// TIA Portal V17 export
// export: Created 2024-09-02T12:50:26.2822455Z, ExportSetting WithDefaults, DisplayName Totally Integrated Automation Portal, DisplayVersion V17, DisplayName TIA Portal Openness, DisplayVersion V17, DisplayName TIA Portal Version Control Interface, DisplayVersion V17, DisplayName STEP 7 Professional, DisplayVersion V17, DisplayName STEP 7 Safety, DisplayVersion V17, DisplayName WinCC Professional, DisplayVersion V17
TYPE "TypeOperatingModes"
// stored: IsFailsafeCompliant false
   STRUCT
      lamp_test : Bool;   // Lampentest / Lamp test
      switchon_conditions_nok : Bool;   // Einschaltbedinnung NIO / Switch-on condition NOK
      Estop_nok : Bool;   // Not-Aus n.i.O. / Emergency stop n. i. O.
      sg_nok : Bool;   // Schutzgitter n.i.O. / Protective grille NOK
      report_contr_nok : Bool;   // Melderkontrolle NIO / Detector control NIO
      startcond_ready : Bool;   // Startvoraussetzungen Bereit / Starting conditions Ready
      start_conditions_on : Bool;   // Startvoraussetzungen sind ein / Starting conditions are ON
      media_on : Bool;   // Medien Ein / Media ON
      mode_auto : Bool;   // Betriebsart Automatik / Operating mode Automatic
      mode_hand : Bool;   // Betriebsart Hand / Operating mode Hand
      start_on : Bool;   // Start Ein / Start On
      tacte_end : Bool;   // Halt Taktende aktiv / Stop Clock end active
      fault_ack : Bool;   // Störung Quittieren / Acknowledge fault
      hm_fault_ack : Array[1..8] of Bool;   // HM Störung Quitt / HM Fault Acknowledge
      sk_fault_ack : Bool;   // Störung Quittieren (SK) / Acknowledge fault (SK)
      "mode_auto+start" : Bool;   // Betriebsart Auto + Start / Operating mode Auto + Start
      "mode_hand+start" : Bool;   // Betriebsart Hand + Start / Manual Operating manual + start
      home_running : Bool;   // Grundstellungsfahrt aktiv / Basic position travel active
      home_activated : Bool;   // Grundstellungstaste betätigt / Basic position button pressed
      home_active : Bool;   // Grundstellungsfahrt wurde aktiviert / Basic position travel has been activated
      protective_circuit_ack : Bool;   // Schutzkreise Quittieren / Acknowledge protective circuits
      f_module_ack : Bool;   // Fehlersichere Baugruppen Quittieren / Acknowledge fail-safe assemblies
      sk_step_sequence : Bool;   // Schrittketten Schrittbetrieb / Step sequence Step operation
      sk_step_sequence_tact : Bool;   // Schrittketten Schrittbetrieb Takten / Step sequence Step mode takt
      mode_service : Bool;   // Betriebsart Service / Operating mode Service
      operating_report : Bool;   // Betriebsmeldung / Operating message
      defect_report : Bool;   // Mangelmeldung / defect report
      error_report : Bool;   // Fehlermeldung Anwender / Alarm User
      error_report_HBT : Bool;   // Fehlermeldung mit HTE / Alarm with HTE
      error_report_SK : Bool;   // Fehlermeldung Schrittkette / Alarm step chain
      error_report_Aut : Bool;   // Fehlermeldung Automatik Start / Alarm Automatic Start
      error_report_present : Bool;   // Fehlermeldung vorhanden / Error message available
      Fault_Nr : Int;   // Anzahl Störungen / Number of faults
      Information_Nr : Int;   // Anzahl Meldungen / Number of messages
      "fl_pos_mode_auto+start" : Bool;   // positive Flanke Auto + Start / positive edge Auto + Start
      "fl_neg_mode_auto+start" : Bool;   // negative Flanke Auto + Start / negative edge Auto + Start
      hm_fl_pos_mode_auto : Bool;   // HM positive Flanke Auto + Start / HM positive edge Auto + Start
      hm_fl_neg_mode_auto : Bool;   // HM negative Flanke Auto + Start / HM negative edge Auto + Start
      machine_home : Bool;   // Grundstellung erreicht / Basic position reached
      all_units_ready : Bool;   // alle Einheiten fertig / All Units finished
      takt_end_position_reached : Bool;   // Haltepunkt fuer Taktende erreicht / Stop for clock end reached
      f_pos_home_running : Bool;   // positive Flanke Grundstellungsfahrt aktiv / positive edge Basic position travel active
      f_neg_home_runnning : Bool;   // negative Flanke Grundstellungsfahrt aktiv / Negative edge basic position travel active
      hm_f_pos_home_running : Bool;   // HM positive Flanke Grundstellungsfahrt aktiv / HM positive edge Basic position travel active
      hm_f_neg_home_runing : Bool;   // HM negative Flanke Grundstellungsfahrt aktiv / HM negative edge Basic position movement active
      f_neg_mode_start_off : Bool;   // negative Flanke Start Aus / negative edge Start Off
      f_pos_mode_start_on : Bool;   // HM2 positive flanke Betriebsartenwechsel / HM2 positive edge operating mode changes
      hm_f_neg_mode_start_off : Bool;   // HM negative Flanke Start aus / HM negative edge Start off
      hm_f_pos_mode_start_on : Bool;   // HM positive Flanke Start ein / HM positive edge Start on
      f_pos_operating_mode : Bool;   // positive Flanke Betriebsart / positive edge Operating mode
      f_hm1_operating_mode : Bool;   // Hilfsmerker Flanke Betriebsart / Auxiliary flag Flank Operating mode
      f_hm2_operating_mode : Bool;   // Hilfsmerker Flanke Betriebsart / Auxiliary flag Flank Operating mode
      hm_start_conditions_on : Bool;   // Hilfsmerker Startvoraussetzungen sind ein / Auxiliary flags Starting conditions are ON
      fp_start_conditions_on : Bool;   // Flanke Startvoraussetzungen sind ein / Flank Starting conditions are ON
      Pulse_fault_ack { S7_SetPoint := 'True'} : TP_TIME;   // Impulszeit Störung quittieren / Pulse time Acknowledge fault
      Pulse_safetycircuit_ack { S7_SetPoint := 'True'} : TP_TIME;   // Impulszeit Schutzkreise quitt / Pulse time Protective circuits acknowledge
      Pulse_sk_fault_ack { S7_SetPoint := 'True'} : TP_TIME;   // Impulszeit Schrittketten Störung quittieren / Pulse time Step sequence Acknowledge fault
      Pulse_startconditions_on { S7_SetPoint := 'True'} : TP_TIME;   // Impulszeit Startvoraussetzungen ein / Pulse time Start conditions on
      Pulse_f_module_ack { S7_SetPoint := 'True'} : TP_TIME;   // Impulszeit F-Baugruppen quittieren / Acknowledge pulse time of F modules
      Pulse_fault_on : Bool;   // Impuls Startvoraussetzungen ein / Impulse Start conditions on
      Delay_Time_control_start_conditions { S7_SetPoint := 'True'} : TON_TIME;   // Verzögerungszeit Überwachung Startvoraussetzungen / Delay time Monitoring Starting conditions
      Delay_control_start_conditions : Bool;   // Verzögerung Überwachung Startvoraussetzungen / Delay Monitoring Starting conditions
      Delay_Time_start_conditions_ok { S7_SetPoint := 'True'} : TON_TIME;   // Verzögerungszeit Startvoraussetzungen IO / Delay time Start conditions OK
      Delay_start_conditions_ok : Bool;   // Verzögerungszeit Startvoraussetzungen IO / Delay time Start conditions OK
      Delay_Time_valve_reset { S7_SetPoint := 'True'} : TON_TIME;   // Verzögerungszeit Ventile Reset / Delay time for valves Reset
      Delay_Time_display_switchon_conditions { S7_SetPoint := 'True'} : TON_TIME;   // Verzögerungszeit Anzeige Fehler Einschaltbedinung / Delay time Display Error Switch-on condition
      Delay_Time_home_reached { S7_SetPoint := 'True'} : TON_TIME;   // Verzögerungszeit GS erreicht / Delay time GS reached
      Delay_home_reached : Bool;   // Verzögerung GS erreicht / Delay Home reached
      Delay_feedback_circuit { S7_SetPoint := 'True'} : Array[1..8] of TON_TIME;   // Verzögerung Störung Rückführkreis / Delay fault feedback loop
      Delay_pneumatic_defect { S7_SetPoint := 'True'} : Array[1..8] of TON_TIME;   // Versögerung Störung Pneumatikdruck abgefallen / Delay Fault Pneumatic pressure droped
      Delay_protection_fault { S7_SetPoint := 'True'} : Array[1..8] of TON_TIME;   // Versögerung Störung Schütz abgefallen / Delay fault contactor dropped out
   END_STRUCT;
END_TYPE
